{attribute addProperty BoxType "EK1100-0000-0018"}
{attribute addProperty Id "Beckhoff_AMI8xxxEK1122Beckhoff_AMI8xxxEK1122_F1A965BF64080"}
{attribute addProperty CRC "2270709332"}
{attribute addProperty SizeInBites "640"}
{attribute addProperty SizeInBytes "80"}
TYPE EK1100_Beckhoff_AMI8xxx_87584654 EXTENDS EK1100_179A0949 :
STRUCT
	{attribute addProperty Name "Beckhoff_AMI8xxxEK1122"}
	Beckhoff_AMI8xxxEK1122 : Beckhoff_AMI8xxxEK1122_F1A965BF;
END_STRUCT
END_TYPE

(* stored: Version 1.2.0.0, ProductVersion 3.1.4024.9
   DUT EK1100_Beckhoff_AMI8xxx_87584654: Id {7452c4b8-c6aa-42da-bf77-c16562fc87ef} *)
